// TIA Portal V20 export
// export: Created 2025-12-01T14:57:26.2869772Z, ExportSetting None, DisplayName Totally Integrated Automation Portal, DisplayVersion V20 Update 3, DisplayName TIA Portal Openness, DisplayVersion V20 Update 3, DisplayName TIA Portal Version Control Interface, DisplayVersion V20 Update 3, DisplayName STEP 7 Professional, DisplayVersion V20 Update 3, DisplayName STEP 7 Safety, DisplayVersion V20 Update 2, DisplayName WinCC Basic/Comfort/Advanced, DisplayVersion V20 Update 3, DisplayName WinCC Professional, DisplayVersion V20 Update 3, DisplayName WinCC Unified, DisplayVersion V20 Update 3
FUNCTION "FC945_Control_BWU4893" : Void   // FC945, SCL
{ S7_Optimized_Access := 'FALSE' }
// stored: AutoNumber false, SetENOAutomatically false
   VAR_INPUT
      numero_tarjeta : Int;
      "2_o_4_motores?" : USInt;
      dir_inicial : Int;
      M1 : Bool;
      M2 : Bool;
      M3 : Bool;
      M4 : Bool;
   END_VAR
   VAR_TEMP
      valor_tmp : UInt;
      cero : SInt;
      retval : Word;
   END_VAR
BEGIN
   // calcular la dirección donde tenemos que recoger los datos para luego escribirlos en periferia

   #valor_tmp := ((#numero_tarjeta - 1) * 28) + 20;

   // borramos los datos convertidos antes de convertir por si hay valores residuales
   // 
   #cero := 0;

   //#retval:=FILL(BVAL := #cero, BLK => "datos_bwu4893".tarjeta[#numero_tarjeta]);

   IF (#"2_o_4_motores?" = 0) OR (#"2_o_4_motores?" > 4) THEN
       RETURN; // no está bien configurado
   END_IF;

       REGION 2_motores
           IF #"2_o_4_motores?" = 2 THEN
               // conversión del dato de la consigna de velocidad de m/min a consigna en %
               // 
               IF #M1 THEN
                   "DB945_Datos_BWU4893".tarjeta[#numero_tarjeta].Consigna_convertida_1 := LIMIT(MN := -100, IN := ROUND(((("DB945_Datos_BWU4893".tarjeta[#numero_tarjeta].consigna_1) / 60.0)) * 100.0), MX := 100);
                   ;
               ELSE
                   "DB945_Datos_BWU4893".tarjeta[#numero_tarjeta].Consigna_convertida_1 := LIMIT(MN := -100, IN := ROUND((((0) / 60.0)) * 100.0), MX := 100);
                   ;
               END_IF;

               IF #M2 THEN
                   "DB945_Datos_BWU4893".tarjeta[#numero_tarjeta].Consigna_convertida_2 := LIMIT(MN := -100, IN := ROUND(((("DB945_Datos_BWU4893".tarjeta[#numero_tarjeta].consigna_2) / 60.0)) * 100.0), MX := 100);
                   ;
               ELSE
                   "DB945_Datos_BWU4893".tarjeta[#numero_tarjeta].Consigna_convertida_2 := LIMIT(MN := -100, IN := ROUND((((0) / 60.0)) * 100.0), MX := 100);
                   ;
               END_IF;



              // "datos_bwu4893".tarjeta[#numero_tarjeta].Consigna_convertida_1 := LIMIT(MN := -100, IN := ROUND(((("datos_bwu4893".tarjeta[#numero_tarjeta].consigna_1) / 60.0)) * 100.0), MX := 100);
              // "datos_bwu4893".tarjeta[#numero_tarjeta].Consigna_convertida_2 := LIMIT(MN := -100, IN := ROUND(((("datos_bwu4893".tarjeta[#numero_tarjeta].consigna_2) / 60.0)) * 100.0), MX := 100);
               "DB945_Datos_BWU4893".tarjeta[#numero_tarjeta].Consigna_convertida_3 := 0;
               "DB945_Datos_BWU4893".tarjeta[#numero_tarjeta].Consigna_convertida_4 := 0;
               // conversión del dato de la rampa de segundos 0--25.5 a %
               // 
               "DB945_Datos_BWU4893".tarjeta[#numero_tarjeta].Rampa_convertida_1 := LIMIT(MN := 0, IN := ROUND((("DB945_Datos_BWU4893".tarjeta[#numero_tarjeta].rampa_1 * 100.0) / 25.5)), MX := 100);
               "DB945_Datos_BWU4893".tarjeta[#numero_tarjeta].Rampa_convertida_2 := LIMIT(MN := 0, IN := ROUND((("DB945_Datos_BWU4893".tarjeta[#numero_tarjeta].rampa_2 * 100.0) / 25.5)), MX := 100);
               "DB945_Datos_BWU4893".tarjeta[#numero_tarjeta].Rampa_convertida_3 := 0;
               "DB945_Datos_BWU4893".tarjeta[#numero_tarjeta].Rampa_convertida_4 := 0;
               // escribir los datos en periferia

               POKE_BLK(area_src := 16#84,
                        dbNumber_src := 945,
                        byteOffset_src := #valor_tmp,
                        area_dest := 16#82,
                        dbNumber_dest := 0,
                        byteOffset_dest := #dir_inicial,
                        count := 2);

               POKE_BLK(area_src := 16#84,
                        dbNumber_src := 945,
                        byteOffset_src := (#valor_tmp + 4),
                        area_dest := 16#82,
                        dbNumber_dest := 0,
                        byteOffset_dest := (#dir_inicial + 2),
                        count := 2);


           END_IF;
       END_REGION
       REGION 4_Motores
           IF (#"2_o_4_motores?" > 2) AND (#"2_o_4_motores?" <= 4) THEN

               // conversión del dato de la consigna de velocidad de m/min a consigna en %


               IF #M1 THEN
                   "DB945_Datos_BWU4893".tarjeta[#numero_tarjeta].Consigna_convertida_1 := LIMIT(MN := -100, IN := ROUND(((("DB945_Datos_BWU4893".tarjeta[#numero_tarjeta].consigna_1) / 60.0)) * 100.0), MX := 100);
                   ;
               ELSE
                   "DB945_Datos_BWU4893".tarjeta[#numero_tarjeta].Consigna_convertida_1 := LIMIT(MN := -100, IN := ROUND((((0) / 60.0)) * 100.0), MX := 100);
                   ;
               END_IF;

               IF #M2 THEN
                   "DB945_Datos_BWU4893".tarjeta[#numero_tarjeta].Consigna_convertida_2 := LIMIT(MN := -100, IN := ROUND(((("DB945_Datos_BWU4893".tarjeta[#numero_tarjeta].consigna_2) / 60.0)) * 100.0), MX := 100);
                   ;
               ELSE
                   "DB945_Datos_BWU4893".tarjeta[#numero_tarjeta].Consigna_convertida_2 := LIMIT(MN := -100, IN := ROUND((((0) / 60.0)) * 100.0), MX := 100);
                   ;
               END_IF;

               IF #M3 THEN
                   "DB945_Datos_BWU4893".tarjeta[#numero_tarjeta].Consigna_convertida_3 := LIMIT(MN := -100, IN := ROUND(((("DB945_Datos_BWU4893".tarjeta[#numero_tarjeta].consigna_3) / 60.0)) * 100.0), MX := 100);
                   ;
               ELSE
                   "DB945_Datos_BWU4893".tarjeta[#numero_tarjeta].Consigna_convertida_3 := LIMIT(MN := -100, IN := ROUND((((0) / 60.0)) * 100.0), MX := 100);
                   ;
               END_IF;

               IF #M4 THEN
                   "DB945_Datos_BWU4893".tarjeta[#numero_tarjeta].Consigna_convertida_4 := LIMIT(MN := -100, IN := ROUND(((("DB945_Datos_BWU4893".tarjeta[#numero_tarjeta].consigna_4) / 60.0)) * 100.0), MX := 100);
                   ;
               ELSE
                   "DB945_Datos_BWU4893".tarjeta[#numero_tarjeta].Consigna_convertida_4 := LIMIT(MN := -100, IN := ROUND((((0) / 60.0)) * 100.0), MX := 100);
                   ;
               END_IF;



             //  "datos_bwu4893".tarjeta[#numero_tarjeta].Consigna_convertida_1 := LIMIT(MN := -100, IN := ROUND(((("datos_bwu4893".tarjeta[#numero_tarjeta].consigna_1) / 60.0)) * 100.0), MX := 100);
             //  "datos_bwu4893".tarjeta[#numero_tarjeta].Consigna_convertida_2 := LIMIT(MN := -100, IN := ROUND(((("datos_bwu4893".tarjeta[#numero_tarjeta].consigna_2) / 60.0)) * 100.0), MX := 100);
             //  "datos_bwu4893".tarjeta[#numero_tarjeta].Consigna_convertida_3 := LIMIT(MN := -100, IN := ROUND(((("datos_bwu4893".tarjeta[#numero_tarjeta].consigna_3) / 60.0)) * 100.0), MX := 100);
             //  "datos_bwu4893".tarjeta[#numero_tarjeta].Consigna_convertida_4 := LIMIT(MN := -100, IN := ROUND(((("datos_bwu4893".tarjeta[#numero_tarjeta].consigna_4) / 60.0)) * 100.0), MX := 100);


               // conversión del dato de la rampa de segundos 0--25.5 a %

               "DB945_Datos_BWU4893".tarjeta[#numero_tarjeta].Rampa_convertida_1 := LIMIT(MN := 0, IN := ROUND((("DB945_Datos_BWU4893".tarjeta[#numero_tarjeta].rampa_1 * 100.0) / 25.5)), MX := 100);
               "DB945_Datos_BWU4893".tarjeta[#numero_tarjeta].Rampa_convertida_2 := LIMIT(MN := 0, IN := ROUND((("DB945_Datos_BWU4893".tarjeta[#numero_tarjeta].rampa_2 * 100.0) / 25.5)), MX := 100);
               "DB945_Datos_BWU4893".tarjeta[#numero_tarjeta].Rampa_convertida_3 := LIMIT(MN := 0, IN := ROUND((("DB945_Datos_BWU4893".tarjeta[#numero_tarjeta].rampa_3 * 100.0) / 25.5)), MX := 100);
               "DB945_Datos_BWU4893".tarjeta[#numero_tarjeta].Rampa_convertida_4 := LIMIT(MN := 0, IN := ROUND((("DB945_Datos_BWU4893".tarjeta[#numero_tarjeta].rampa_4 * 100.0) / 25.5)), MX := 100);


               // escribir los datos en periferia

               POKE_BLK(area_src := 16#84,
                        dbNumber_src := 945,
                        byteOffset_src := #valor_tmp,
                        area_dest := 16#82,
                        dbNumber_dest := 0,
                        byteOffset_dest := #dir_inicial,
                        count := 8);



           END_IF;
       END_REGION
END_FUNCTION
